PROGRAM crosswalkErrorChecks
VAR
END_VAR
VAR // added by the converter: edge detectors and wires of the graphical bodies
    _w1, _w2, _w3, _w4 : BOOL;
END_VAR

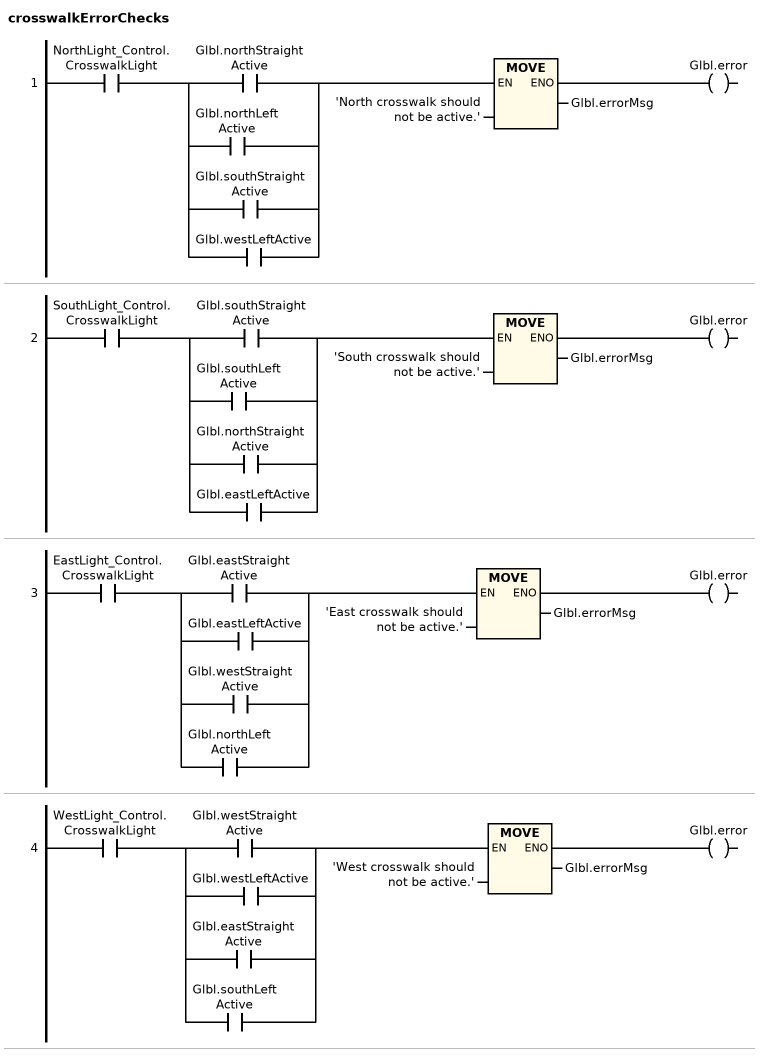
// NETWORK 1
_w1 := NorthLight_Control.CrosswalkLight AND (Glbl.northStraightActive OR Glbl.northLeftActive OR Glbl.southStraightActive OR Glbl.westLeftActive);
IF _w1 THEN Glbl.errorMsg := 'North crosswalk should not be active.'; END_IF
Glbl.error := _w1;

// NETWORK 2
_w2 := SouthLight_Control.CrosswalkLight AND (Glbl.southStraightActive OR Glbl.southLeftActive OR Glbl.northStraightActive OR Glbl.eastLeftActive);
IF _w2 THEN Glbl.errorMsg := 'South crosswalk should not be active.'; END_IF
Glbl.error := _w2;

// NETWORK 3
_w3 := EastLight_Control.CrosswalkLight AND (Glbl.eastStraightActive OR Glbl.eastLeftActive OR Glbl.westStraightActive OR Glbl.northLeftActive);
IF _w3 THEN Glbl.errorMsg := 'East crosswalk should not be active.'; END_IF
Glbl.error := _w3;

// NETWORK 4
_w4 := WestLight_Control.CrosswalkLight AND (Glbl.westStraightActive OR Glbl.westLeftActive OR Glbl.eastStraightActive OR Glbl.southLeftActive);
IF _w4 THEN Glbl.errorMsg := 'West crosswalk should not be active.'; END_IF
Glbl.error := _w4;

END_PROGRAM

(* stored: Version 1.1.0.1, ProductVersion 3.1.4022.10
   POU crosswalkErrorChecks: Id {a9e4090f-8a2c-4e93-9f09-e71f0371e42c}, SpecialFunc None *)
